TYPE ST_VC_AccessPanel :
STRUCT
	inputs : ST_VC_AccessPanelInputs;
	outputs : ST_VC_AccessPanelOutputs;
END_STRUCT
END_TYPE

(* stored: Version 1.1.0.1, ProductVersion 3.1.4024.9
   DUT ST_VC_AccessPanel: Id {06a8cd1b-1db3-40b4-86b4-aea408f7bb47} *)
